{attribute 'no_explicit_call' := 'do not call this function block directly'} 
FUNCTION_BLOCK ListOfValues EXTENDS GenericList
VAR
	_ClassName : STRING := __POUNAME();
END_VAR

METHOD AppendBool : DINT
VAR_INPUT
	value : BOOL;
END_VAR
AppendBool := Append(value);
END_METHOD

METHOD AppendByte : DINT
VAR_INPUT
	value : BYTE;
END_VAR
AppendByte := Append(value);
END_METHOD

METHOD AppendDate : DINT
VAR_INPUT
	value : DATE;
END_VAR
AppendDate := Append(value);
END_METHOD

METHOD AppendDateAndTime : DINT
VAR_INPUT
	value : DATE_AND_TIME;
END_VAR
AppendDateAndTime := Append(value);
END_METHOD

METHOD AppendDInt : DINT
VAR_INPUT
	value : DINT;
END_VAR
AppendDInt := Append(value);
END_METHOD

METHOD AppendDWord : DINT
VAR_INPUT
	value : DWORD;
END_VAR
AppendDWord := Append(value);
END_METHOD

METHOD AppendInt : DINT
VAR_INPUT
	value : INT;
END_VAR
AppendInt := Append(value);
END_METHOD

METHOD AppendLDate : DINT
VAR_INPUT
	value : LDATE;
END_VAR
AppendLDate := Append(value);
END_METHOD

METHOD AppendLDateAndTime : DINT
VAR_INPUT
	value : LDATE_AND_TIME;
END_VAR
AppendLDateAndTime := Append(value);
END_METHOD

METHOD AppendLInt : DINT
VAR_INPUT
	value : LINT;
END_VAR
AppendLInt := Append(value);
END_METHOD

METHOD AppendLReal : DINT
VAR_INPUT
	value : LREAL;
END_VAR
AppendLReal := Append(value);
END_METHOD

METHOD AppendLTime : DINT
VAR_INPUT
	value : LTIME;
END_VAR
AppendLTime := Append(value);
END_METHOD

METHOD AppendLTimeOfDay : DINT
VAR_INPUT
	value : LTIME_OF_DAY;
END_VAR
AppendLTimeOfDay := Append(value);
END_METHOD

METHOD AppendLWord : DINT
VAR_INPUT
	value : LWORD;
END_VAR
AppendLWord := Append(value);
END_METHOD

METHOD AppendObject : DINT
VAR_INPUT
	value : IObject;
	owningMemory : BOOL;
END_VAR
VAR
	genericValue : GENERIC_VALUE;
END_VAR
genericValue.FromObject(value, TRUE);

AppendObject := AppendGenericValue(genericValue);
END_METHOD

METHOD AppendReal : DINT
VAR_INPUT
	value : REAL;
END_VAR
AppendReal := Append(value);
END_METHOD

METHOD AppendSInt : DINT
VAR_INPUT
	value : SINT;
END_VAR
AppendSInt := Append(value);
END_METHOD

METHOD AppendString : DINT
VAR_IN_OUT CONSTANT
	value : STRING;
END_VAR
VAR
	genericValue : GENERIC_VALUE;
END_VAR
genericValue.FromAnyType(StringHelper.StringPointerToAnyType(ADR(value)), StoredTypeCategory = TYPE_CATEGORY.VALUE_TYPE, TRUE);

AppendString := AppendGenericValue(genericValue);
END_METHOD

METHOD AppendTime : DINT
VAR_INPUT
	value : TIME;
END_VAR
AppendTime := Append(value);
END_METHOD

METHOD AppendTimeOfDay : DINT
VAR_INPUT
	value : TIME_OF_DAY;
END_VAR
AppendTimeOfDay := Append(value);
END_METHOD

METHOD AppendUDInt : DINT
VAR_INPUT
	value : UDINT;
END_VAR
AppendUDInt := Append(value);
END_METHOD

METHOD AppendUInt : DINT
VAR_INPUT
	value : UINT;
END_VAR
AppendUInt := Append(value);
END_METHOD

METHOD AppendULInt : DINT
VAR_INPUT
	value : ULINT;
END_VAR
AppendULInt := Append(value);
END_METHOD

METHOD AppendUSInt : DINT 
VAR_INPUT
	value : USINT;
END_VAR
AppendUSInt := Append(value);
END_METHOD

METHOD AppendWord : DINT 
VAR_INPUT
	value : WORD;
END_VAR
AppendWord := Append(value);
END_METHOD

METHOD AppendWString : DINT
VAR_IN_OUT CONSTANT
	value : WSTRING(255);
END_VAR
VAR
	genericValue : GENERIC_VALUE;
END_VAR
genericValue.FromAnyType(WideStringHelper.StringPointerToAnyType(ADR(value)), StoredTypeCategory = TYPE_CATEGORY.VALUE_TYPE, TRUE);

AppendWString := AppendGenericValue(genericValue);
END_METHOD

{attribute 'monitoring' := 'call'}
PROPERTY ClassName : STRING
GET
ClassName := _ClassName;
END_GET
END_PROPERTY

METHOD FB_init : BOOL
VAR_INPUT
	(* if TRUE, the retain variables are initialized (warm start / cold start)*)
	bInitRetains	: BOOL;
	(* if TRUE, the instance afterwards gets moved into the copy code (online change)*)
	bInCopyCode	: BOOL;
END_VAR
StoredTypeCategory := TYPE_CATEGORY.VALUE_TYPE;
END_METHOD

METHOD InsertBool 
VAR_INPUT
	value : BOOL;
	index : DINT;
END_VAR
Insert(value, index);
END_METHOD

METHOD InsertByte 
VAR_INPUT
	value : BYTE;
	index : DINT;
END_VAR
Insert(value, index);
END_METHOD

METHOD InsertDate 
VAR_INPUT
	value : DATE;
	index : DINT;
END_VAR
Insert(value, index);
END_METHOD

METHOD InsertDateAndTime 
VAR_INPUT
	value : DATE_AND_TIME;
	index : DINT;
END_VAR
Insert(value, index);
END_METHOD

METHOD InsertDInt 
VAR_INPUT
	value : DINT;
	index : DINT;
END_VAR
Insert(value, index);
END_METHOD

METHOD InsertDWord 
VAR_INPUT
	value : DWORD;
	index : DINT;
END_VAR
Insert(value, index);
END_METHOD

METHOD InsertInt 
VAR_INPUT
	value : INT;
	index : DINT;
END_VAR
Insert(value, index);
END_METHOD

METHOD InsertLDate 
VAR_INPUT
	value : LDATE;
	index : DINT;
END_VAR
Insert(value, index);
END_METHOD

METHOD InsertLDateAndTime 
VAR_INPUT
	value : LDATE_AND_TIME;
	index : DINT;
END_VAR
Insert(value, index);
END_METHOD

METHOD InsertLInt 
VAR_INPUT
	value : LINT;
	index : DINT;
END_VAR
Insert(value, index);
END_METHOD

METHOD InsertLReal 
VAR_INPUT
	value : LREAL;
	index : DINT;
END_VAR
Insert(value, index);
END_METHOD

METHOD InsertLTime 
VAR_INPUT
	value : LTIME;
	index : DINT;
END_VAR
Insert(value, index);
END_METHOD

METHOD InsertLTimeOfDay 
VAR_INPUT
	value : LTIME_OF_DAY;
	index : DINT;
END_VAR
Insert(value, index);
END_METHOD

METHOD InsertLWord 
VAR_INPUT
	value : LWORD;
	index : DINT;
END_VAR
Insert(value, index);
END_METHOD

METHOD InsertObject 
VAR_INPUT
	value : IObject;
	index : DINT;
END_VAR
VAR
	genericValue : GENERIC_VALUE;
END_VAR
genericValue.FromObject(value, TRUE);

InsertGenericValue(genericValue, index);
END_METHOD

METHOD InsertReal 
VAR_INPUT
	value : REAL;
	index : DINT;
END_VAR
Insert(value, index);
END_METHOD

METHOD InsertSInt 
VAR_INPUT
	value : SINT;
	index : DINT;
END_VAR
Insert(value, index);
END_METHOD

METHOD InsertString 
VAR_IN_OUT CONSTANT
	value : STRING;
END_VAR
VAR_INPUT
	index : DINT;
END_VAR
VAR
	genericValue : GENERIC_VALUE;
END_VAR
genericValue.FromAnyType(StringHelper.StringPointerToAnyType(ADR(value)), StoredTypeCategory = TYPE_CATEGORY.VALUE_TYPE, TRUE);

InsertGenericValue(genericValue, index);
END_METHOD

METHOD InsertTime 
VAR_INPUT
	value : TIME;
	index : DINT;
END_VAR
Insert(value, index);
END_METHOD

METHOD InsertTimeOfDay 
VAR_INPUT
	value : TIME_OF_DAY;
	index : DINT;
END_VAR
Insert(value, index);
END_METHOD

METHOD InsertUDInt 
VAR_INPUT
	value : UDINT;
	index : DINT;
END_VAR
Insert(value, index);
END_METHOD

METHOD InsertUInt 
VAR_INPUT
	value : UINT;
	index : DINT;
END_VAR
Insert(value, index);
END_METHOD

METHOD InsertULInt 
VAR_INPUT
	value : ULINT;
	index : DINT;
END_VAR
Insert(value, index);
END_METHOD

METHOD InsertUSInt 
VAR_INPUT
	value : USINT;
	index : DINT;
END_VAR
Insert(value, index);
END_METHOD

METHOD InsertWord 
VAR_INPUT
	value : WORD;
	index : DINT;
END_VAR
Insert(value, index);
END_METHOD

METHOD InsertWString 
VAR_IN_OUT CONSTANT
	value : WSTRING;
END_VAR
VAR_INPUT
	index : DINT;
END_VAR
VAR
	genericValue : GENERIC_VALUE;
END_VAR
genericValue.FromAnyType(WideStringHelper.StringPointerToAnyType(ADR(value)), StoredTypeCategory = TYPE_CATEGORY.VALUE_TYPE, TRUE);

InsertGenericValue(genericValue, index);
END_METHOD

METHOD SetBool
VAR_INPUT
	value : BOOL;
	index : DINT;
END_VAR
Set(value, index, FALSE);
END_METHOD

METHOD SetByte
VAR_INPUT
	value : BYTE;
	index : DINT;
END_VAR
Set(value, index, FALSE);
END_METHOD

METHOD SetDate
VAR_INPUT
	value : DATE;
	index : DINT;
END_VAR
Set(value, index, FALSE);
END_METHOD

METHOD SetDateAndTime
VAR_INPUT
	value : DATE_AND_TIME;
	index : DINT;
END_VAR
Set(value, index, FALSE);
END_METHOD

METHOD SetDInt
VAR_INPUT
	value : DINT;
	index : DINT;
END_VAR
Set(value, index, FALSE);
END_METHOD

METHOD SetDWord
VAR_INPUT
	value : DWORD;
	index : DINT;
END_VAR
Set(value, index, FALSE);
END_METHOD

METHOD SetInt
VAR_INPUT
	value : INT;
	index : DINT;
END_VAR
Set(value, index, FALSE);
END_METHOD

METHOD SetLDate
VAR_INPUT
	value : LDATE;
	index : DINT;
END_VAR
Set(value, index, FALSE);
END_METHOD

METHOD SetLDateAndTime
VAR_INPUT
	value : LDATE_AND_TIME;
	index : DINT;
END_VAR
Set(value, index, FALSE);
END_METHOD

METHOD SetLInt
VAR_INPUT
	value : LINT;
	index : DINT;
END_VAR
Set(value, index, FALSE);
END_METHOD

METHOD SetLReal
VAR_INPUT
	value : LREAL;
	index : DINT;
END_VAR
Set(value, index, FALSE);
END_METHOD

METHOD SetLTime
VAR_INPUT
	value : LTIME;
	index : DINT;
END_VAR
Set(value, index, FALSE);
END_METHOD

METHOD SetLTimeOfDay
VAR_INPUT
	value : LTIME_OF_DAY;
	index : DINT;
END_VAR
Set(value, index, FALSE);
END_METHOD

METHOD SetLWord
VAR_INPUT
	value : LWORD;
	index : DINT;
END_VAR
Set(value, index, FALSE);
END_METHOD

METHOD SetObject
VAR_INPUT
	value : IObject;
	index : DINT;
END_VAR
VAR
	genericValue : GENERIC_VALUE;
END_VAR
genericValue.FromObject(value, TRUE);

SetGenericValue(genericValue, index);
END_METHOD

METHOD SetReal
VAR_INPUT
	value : REAL;
	index : DINT;
END_VAR
Set(value, index, FALSE);
END_METHOD

METHOD SetSInt
VAR_INPUT
	value : SINT;
	index : DINT;
END_VAR
Set(value, index, FALSE);
END_METHOD

METHOD SetString
VAR_IN_OUT CONSTANT
	value : STRING;
END_VAR
VAR_INPUT
	index : DINT;
END_VAR
VAR
	genericValue : GENERIC_VALUE;
END_VAR
genericValue.FromAnyType(StringHelper.StringPointerToAnyType(ADR(value)), StoredTypeCategory = TYPE_CATEGORY.VALUE_TYPE, TRUE);

SetGenericValue(genericValue, index);
END_METHOD

METHOD SetTime
VAR_INPUT
	value : TIME;
	index : DINT;
END_VAR
Set(value, index, FALSE);
END_METHOD

METHOD SetTimeOfDay
VAR_INPUT
	value : TIME_OF_DAY;
	index : DINT;
END_VAR
Set(value, index, FALSE);
END_METHOD

METHOD SetUDInt
VAR_INPUT
	value : UDINT;
	index : DINT;
END_VAR
Set(value, index, FALSE);
END_METHOD

METHOD SetUInt
VAR_INPUT
	value : UINT;
	index : DINT;
END_VAR
Set(value, index, FALSE);
END_METHOD

METHOD SetULInt
VAR_INPUT
	value : ULINT;
	index : DINT;
END_VAR
Set(value, index, FALSE);
END_METHOD

METHOD SetUSInt
VAR_INPUT
	value : USINT;
	index : DINT;
END_VAR
Set(value, index, FALSE);
END_METHOD

METHOD SetWord
VAR_INPUT
	value : WORD;
	index : DINT;
END_VAR
Set(value, index, FALSE);
END_METHOD

METHOD SetWString
VAR_IN_OUT CONSTANT
	value : STRING;
END_VAR
VAR_INPUT
	index : DINT;
END_VAR
VAR
	genericValue : GENERIC_VALUE;
END_VAR
genericValue.FromAnyType(WideStringHelper.StringPointerToAnyType(ADR(value)), StoredTypeCategory = TYPE_CATEGORY.VALUE_TYPE, TRUE);

SetGenericValue(genericValue, index);
END_METHOD

END_FUNCTION_BLOCK

(* stored: Version 1.1.0.1
   POU ListOfValues: Id {221bbc0d-e247-4e75-b77f-cd91d2b94914}, SpecialFunc None
   Folder FromTyped: Id {acd1b00a-3231-43e3-86b5-9cb6372d5cd9}
   Folder Bool: Id {9090178e-9b01-4482-9588-96e251e64575}
   Folder Date and time: Id {5eefb26a-d859-4fd5-81be-8985db57b358}
   Folder Date: Id {5ebfa31c-736b-4ae3-ad18-b998aabba03c}
   Folder DateAndTime: Id {83f0a04d-fd5f-4c99-aa51-2eefb2772047}
   Folder LDate: Id {b544d02c-f87a-441d-980a-4d286e46fa86}
   Folder LDateAndTime: Id {88a7e84f-f34d-4378-a54f-dc3e887cc691}
   Folder LTime: Id {60738d7d-6ca0-4029-8281-0615b999384f}
   Folder LTimeOfDay: Id {0a7aead2-359e-433d-960f-0c10693d7224}
   Folder Time: Id {38274cb0-8364-45eb-8e88-215e28cc42b3}
   Folder TimeOfDay: Id {7d17033c-d4a4-4c13-af60-f2ed7191ea27}
   Folder Floating point: Id {fe8f5428-c58c-403b-a822-f316c2d2d305}
   Folder LReal: Id {1b7f625c-aee1-42a4-9543-e172d975e6d6}
   Folder Real: Id {2c5d86ab-a2ea-4eb8-a6d6-205d80e70b6b}
   Folder Integer: Id {26052080-a976-4f8b-a494-9bb5e6908de8}
   Folder Signed: Id {9d9fc300-427c-4975-a909-58f379899b3c}
   Folder DInt: Id {d55a52fa-7cb9-4126-aa82-a54ac8b907e0}
   Folder Int: Id {945961f1-824b-435c-950d-ea6b0f7d889a}
   Folder LInt: Id {5551eefd-884e-4c30-8010-b766ffee9069}
   Folder SInt: Id {708e760f-e764-4d00-9a56-3638c39d770b}
   Folder Unsugned: Id {1e5b97ac-950c-43d4-b732-c4da17064b87}
   Folder Byte: Id {60bf043d-706f-49ba-b2a2-a82461d1aa6d}
   Folder DWord: Id {23147428-fd27-4475-8165-077c2da0ebf1}
   Folder LWord: Id {943443a3-06af-477b-8f36-afe5703b05e0}
   Folder UDInt: Id {13310a81-de10-4077-aa66-2f666c0ec4a2}
   Folder UInt: Id {96b53809-ad95-43b9-8b54-83398f555442}
   Folder ULInt: Id {55d93a7d-d145-437e-9a1d-de07558e5c67}
   Folder USInt: Id {44a1b581-acce-4374-9426-ce05e5e0026e}
   Folder Word: Id {4f384c28-32aa-4df3-96c4-17b4cc3f45f7}
   Folder Object: Id {1febbf70-e193-417d-96d5-3bd824486127}
   Folder Strings: Id {6bddd30f-89af-41dc-bab0-ba9f9794dcc4}
   Folder String: Id {95c874ac-3bff-45ba-8f40-979386260391}
   Folder WString: Id {bde5aedb-1079-47f5-ac6b-5620e19c6274}
   Method AppendBool: Id {51108fd9-4c0f-4e8b-93e0-2397e67bb007}
   Method AppendByte: Id {ba1a40d8-6582-4812-be2f-b4c7b7475ab0}
   Method AppendDate: Id {3705ade3-8682-4017-b578-13e6b81d3e81}
   Method AppendDateAndTime: Id {53f37d37-fade-4c2c-8ecf-e595eaafdc92}
   Method AppendDInt: Id {1b7e4d63-65fa-4b97-8a90-801dc02a248f}
   Method AppendDWord: Id {0df1b89d-0697-4d45-8b71-8708834a98b8}
   Method AppendInt: Id {8a38a489-1d86-436a-af69-217a564d81d7}
   Method AppendLDate: Id {db98c1ca-d447-4c4c-ac49-e25fd3721f83}
   Method AppendLDateAndTime: Id {c5c8a7a5-0f34-4a75-aa66-d9cb877f1fa1}
   Method AppendLInt: Id {0c5a1d4a-8c17-4b8d-97ec-ceb5eadfee7f}
   Method AppendLReal: Id {d603cc3d-ab4a-440e-9556-390c08def90e}
   Method AppendLTime: Id {9701afe1-6db9-4f1c-9ebc-2f3ffca16192}
   Method AppendLTimeOfDay: Id {2e21c1d2-ea13-4aeb-bb13-40e594f56202}
   Method AppendLWord: Id {7d31767d-77d6-4582-861e-9771c0c85c77}
   Method AppendObject: Id {529ff2b0-d2a5-4181-9b5d-ad91c0e6543f}
   Method AppendReal: Id {635c1331-7dfe-4228-8341-86c71adbd7df}
   Method AppendSInt: Id {e0df5e52-35e1-4d8f-aa99-b79e269a6ca2}
   Method AppendString: Id {dc486ddc-b554-48e5-b2d8-9c7e295c426b}
   Method AppendTime: Id {d7681414-19a1-40d8-94f8-b95a9b28acff}
   Method AppendTimeOfDay: Id {1e9e5afb-6764-44fe-b398-163e02bb18a8}
   Method AppendUDInt: Id {95d8e1d6-3c56-41f6-a1d5-c6f62e471df2}
   Method AppendUInt: Id {085a0312-aa3c-4ecf-97d3-90944bb9e2dc}
   Method AppendULInt: Id {874e80c6-6b7e-4915-8515-3f45cd3f9c36}
   Method AppendUSInt: Id {2e8e3eb2-58bd-4ad4-aadc-221194d65aee}
   Method AppendWord: Id {62483313-944c-45a7-b8ea-12901d8f70c0}
   Method AppendWString: Id {0dcc1d9c-6422-478f-8104-ca8a1714e2ab}
   Property ClassName: Id {45471103-049d-4781-9740-44a79e4f4cd7}
   Get Get: Id {19bff5aa-4df4-4314-8815-2f7f99833682}
   Method FB_init: Id {9c3e0f76-6b59-41e8-89e6-f069c49edaa3}
   Method InsertBool: Id {4040b74e-c516-4093-8879-8d9c4c2d73f3}
   Method InsertByte: Id {228d39d2-1548-4d3b-98a5-6cde01348603}
   Method InsertDate: Id {50b62bc2-4538-40dc-b086-444b2485dcf1}
   Method InsertDateAndTime: Id {d433ad1c-0e02-45c5-9042-b9cfe2b963bb}
   Method InsertDInt: Id {475684f4-f980-43ad-83ca-477232b8b871}
   Method InsertDWord: Id {663df9e8-ec01-4a96-89af-5c6522ad3a3f}
   Method InsertInt: Id {03fa1160-938d-438c-bebb-fdf422c16339}
   Method InsertLDate: Id {d2e402be-b974-49d8-871c-39a1eaa8ebab}
   Method InsertLDateAndTime: Id {c71dbbff-2655-4639-a044-ba3b0e598f3f}
   Method InsertLInt: Id {e9d4ab25-a065-4a0a-8e38-a75e5a0fc518}
   Method InsertLReal: Id {77424e17-158b-4150-9b10-ba03a8711da8}
   Method InsertLTime: Id {b524e291-c2ed-491a-9810-660241e30699}
   Method InsertLTimeOfDay: Id {c41a687c-4202-4ebc-a1ce-c97171253474}
   Method InsertLWord: Id {01957b84-5044-4827-8c70-b3f1afb10fb8}
   Method InsertObject: Id {a2a397fd-a7d8-42e7-92d6-868e376beeac}
   Method InsertReal: Id {d2475465-d77d-45a3-9a20-f279a298525d}
   Method InsertSInt: Id {a76d5ebd-b8cb-476e-8d10-6b69ab1eada3}
   Method InsertString: Id {89f2aecf-ec01-4524-8de7-a3b017d252b9}
   Method InsertTime: Id {aac2cc72-c0d7-4a53-9e81-b3d63a179c35}
   Method InsertTimeOfDay: Id {db7ee9c2-3ba1-4e90-8143-9ba1824a9b9f}
   Method InsertUDInt: Id {c091c015-1b94-4f81-8e01-e5ff7d977500}
   Method InsertUInt: Id {ab96baad-a58e-4fa2-8f01-e12f93e449e7}
   Method InsertULInt: Id {9e66eab2-491d-4941-83fe-341d25036b09}
   Method InsertUSInt: Id {46b8ea25-c348-4449-b3dd-3787739fd719}
   Method InsertWord: Id {50573f68-ed66-4457-acae-308fbc7594da}
   Method InsertWString: Id {7a4126e5-5b64-432f-9563-9de221df3677}
   Method SetBool: Id {e53f8061-8e11-4c00-953b-feb900df26cb}
   Method SetByte: Id {dd2c24e4-8ac6-4325-873d-c7454f762544}
   Method SetDate: Id {f4a744db-e0a0-4c33-bb14-cb4c3b7848fa}
   Method SetDateAndTime: Id {7afd1772-485f-4ddd-86fa-25af0c115076}
   Method SetDInt: Id {52d49887-6506-42ef-ae51-87096ba02c4f}
   Method SetDWord: Id {262b2eca-d502-48d2-8d4b-d20953b6da88}
   Method SetInt: Id {49ed6f86-c597-4b01-b8eb-b46238f2d1a4}
   Method SetLDate: Id {1a49e5f8-727c-4f6f-9ba2-d6c3f270314a}
   Method SetLDateAndTime: Id {3f3f5e34-408c-442d-a044-f8935ce1d566}
   Method SetLInt: Id {3665c438-2d01-4cac-940e-e9b9905bf9c3}
   Method SetLReal: Id {fb45f6a4-5618-4cb4-bf36-c1e2e1558716}
   Method SetLTime: Id {b8cc7ded-ba18-49c2-8989-ebb89295d65b}
   Method SetLTimeOfDay: Id {85c977bf-7779-4d3e-9aad-21a14d1b203f}
   Method SetLWord: Id {b54bedd9-1927-483d-8675-3911bc3f265b}
   Method SetObject: Id {1b8103c2-6070-4eb9-bf71-6e1551469b9f}
   Method SetReal: Id {731c57dc-3a08-4f7d-b2df-9a1f13a4d5a0}
   Method SetSInt: Id {b7ae8f53-06b1-475c-95eb-8efb05380427}
   Method SetString: Id {d6a7bb9d-ea16-4460-8d4c-e8b2552b0b67}
   Method SetTime: Id {300ee8b9-811e-40a2-bd59-1e5bc5d0807b}
   Method SetTimeOfDay: Id {26f65179-4a6d-4175-9be2-a4ba87d27afe}
   Method SetUDInt: Id {a45caf7c-661c-46f5-8d46-04063fdf25f0}
   Method SetUInt: Id {41f1edf1-5079-43a4-90de-8c20d3f7087d}
   Method SetULInt: Id {1cee986b-16c0-49cd-9bd0-2bc08c270da6}
   Method SetUSInt: Id {8c2ca0cb-981d-4c13-8271-e2f8b08eecc7}
   Method SetWord: Id {88aadc2f-5206-4f60-9617-bd51f4d16b4e}
   Method SetWString: Id {64701b5b-2fab-4688-9603-787437d49407} *)
